Staubli VAL3: start.pgx

program start()
begin
  resetMotion()
  movej(jStart, tBroche, mRapide100On)

  call Poche(pStartUsinage, nDiametreFraise, 7, 4, 100, 50, 20)

  movej(jChangeOutil, tBroche, mRapide100On)
  waitEndMove()
end
